FUNCTION_BLOCK FB_TcpIPClient
VAR_INPUT
END_VAR
VAR_OUTPUT
END_VAR
VAR
END_VAR

END_FUNCTION_BLOCK

(* stored: Version 1.1.0.1, ProductVersion 3.1.4026.18
   POU FB_TcpIPClient: Id {e21410d2-9a53-4078-be72-54a1cccf9a2c}, SpecialFunc None *)
